// TIA Portal V16 export
// export: Created 2021-06-17T11:14:33.5982322Z, ExportSetting WithDefaults, DisplayName Totally Integrated Automation Portal, DisplayVersion V16 Update 4, DisplayName TIA Portal Version Control Interface, DisplayVersion V16 Update 2, DisplayName TIA Portal Openness, DisplayVersion V16 Update 4, DisplayName SINAMICS Startdrive Advanced, DisplayVersion V16 Update 5, DisplayName SINAMICS Startdrive G130, G150, S120, S150, SINAMICS MV, S210, DisplayVersion V16 Update 5, DisplayName SINAMICS Startdrive G110M, G120, G120C, G120D, G120P, G115D, DisplayVersion V16 Update 5, DisplayName STEP 7 Professional, DisplayVersion V16 Update 4, DisplayName SIMATIC Energy Suite, DisplayVersion V16 Update 4, DisplayName STEP 7 Safety, DisplayVersion V16, DisplayName WinCC Advanced / Unified PC, DisplayVersion V16 Update 4, DisplayName SIMATIC Visualization Architect, DisplayVersion V16 Update 1
TYPE "Mode"
// stored: IsFailsafeCompliant false
   STRUCT
      Independent { ExternalAccessible := 'False'; ExternalVisible := 'False'; ExternalWritable := 'False'} : Bool := TRUE;   // 1 = Незалежний режим роботи - режими перемикаються як оператором так і командами CmdAuto/Global // 0 = режими перемикаються тільки командами CmdAuto/Global
      Disable { ExternalAccessible := 'False'; ExternalVisible := 'False'; ExternalWritable := 'False'} : Bool;   // 1 = Відключено/Виведено із експлуатації Function change to Stop mode
      Auto { ExternalAccessible := 'False'; ExternalVisible := 'False'; ExternalWritable := 'False'} : Bool := FALSE;   // 1 = Automatic mode Control - controlled via the CmdAuto...
      ManualRemote { ExternalAccessible := 'False'; ExternalVisible := 'False'; ExternalWritable := 'False'} : Bool := TRUE;   // 1 = Manual Remote control mode - ручний дистанційний режим керування із HMI
      ManualLocal { ExternalAccessible := 'False'; ExternalVisible := 'False'; ExternalWritable := 'False'} : Bool;   // 1 = Manual Local control mode - ручний місцевий режим зі щита кнопками
      Service { ExternalAccessible := 'False'; ExternalVisible := 'False'; ExternalWritable := 'False'} : Bool;   // 1 = Сервіс-Сontrol via HMI and no display of errors and warnings
      Repair { ExternalAccessible := 'False'; ExternalVisible := 'False'; ExternalWritable := 'False'} : Bool;   // 1 = Ремонт-No control is possible and no display of errors and warnings
      Simulation { ExternalAccessible := 'False'; ExternalVisible := 'False'; ExternalWritable := 'False'} : Bool;   // 1 = Симуляція - команди на фізичні виходи не передаються - входи/аварії/блокування активуються вручну
      Different { ExternalAccessible := 'False'; ExternalVisible := 'False'; ExternalWritable := 'False'} : Bool;   // (для групи) 1 = різні режими у обєктів групи
   END_STRUCT;
END_TYPE
